KUKA KRL program: TPadraoSTR.src, TPadraoSTR.dat

--- TPadraoSTR.src ---
&ACCESS RV2
DEF TPadraoSTR ( )

   ;FOLD Variaveis Default da Matriz de Pontos
      FOR I = 1 to MaxMatrizI
         FOR J = 1 to MaxMatrizJ
            FOR k = 1 to MaxMatrizK
               Ponto_STR[I,J,k].IndexacaoHorizontal = FALSE
               Ponto_STR[I,J,k].NumCaixas = 0
               Ponto_STR[I,J,k].PickOp = 0
               Ponto_STR[I,J,k].ConfGarraOp = 0
               Ponto_STR[I,J,k].FechaGarraOp = 0
               Ponto_STR[I,J,k].AbreGarraOp = 0
               Ponto_STR[I,J,k].SkipGoHome = FALSE
               Ponto_STR[I,J,k].SkipSobeRelAtual = FALSE
               Ponto_STR[I,J,k].SensoresCaixa = 123456
               Ponto_STR[I,J,k].TravaGarra = False
               Ponto_STR[I,J,k].XApp1Place = DefaultPoint
               Ponto_STR[I,J,k].XApp2Place = DefaultPoint
               Ponto_STR[I,J,k].XPlace = DefaultPoint
               Ponto_STR[I,J,k].OffsetPlace = {x 0,Y 0,Z 0,A 0,B 0,C 0}
            ENDFOR
         ENDFOR
      ENDFOR
   ;ENDFOLD

   ;FOLD Variaveis Default Receita
      FOR I = 1 to MaxReceitas
         Receita_STR[I].PlacesCamada = 1
         Receita_STR[I].Camadas = 1
         Receita_STR[I].AlturaCaixa = 1
         Receita_STR[I].Layers = 1
         Receita_STR[I].OffsetProduto = {x 0,Y 0,Z 0,A 0,B 0,C 0}
         FOR J = 1 to MaxCamadas
            Receita_STR_Layer[I,J] = 1
         ENDFOR
      ENDFOR
   ;ENDFOLD

   ;FOLD Variaveis Default Pallet
      FOR I = 1 to MaxPallets
         Pallet_STR[I].Livre = TRUE
         Pallet_STR[I].Completo = FALSE
         Pallet_STR[I].ReceitaAtual = 1
         Pallet_STR[I].PlaceAtual = 1
         Pallet_STR[I].CamadaAtual = 1
         Pallet_STR[I].BasePoint = {x 0,Y 0,Z 0,A 0,B 0,C 0}
         Pallet_STR[I].OffSetPallet = {x 0,Y 0,Z 0,A 0,B 0,C 0}
      ENDFOR
   ;ENDFOLD

   ;FOLD OffsetEsteira
      OffsetEsteira1 = NULLFRAME
      OffsetEsteira2 = NULLFRAME
      BaseEsteira1 = NULLFRAME
      BaseEsteira1 = NULLFRAME
   ;ENDFOLD

   ;FOLD Principais variaveis
      PalletAtual = 1
      LayerAtual = 1
      PlaceLayerAtual = 1
      ReceitaAtual = 1
      PlaceAtual = 1
      CamadaAtual = 1
   ;ENDFOLD

END

--- TPadraoSTR.dat ---
&ACCESS RV2
DEFDAT TPadraoSTR
   INT  I,J,k
ENDDAT
